// TIA Portal V18 export
TYPE "LGasp_typeBufferQuote"
// stored: IsFailsafeCompliant false
   STRUCT
      ID : DInt;
      n_piece : DInt;   // numero del pezzo a cui fa riferimento la quota
      general : "LGasp_typeArticoloGenerale";
      quota : "LGasp_typeQuota";
      quotaordinata : Bool;   // Quota ordinata da algoritmo riordino
   END_STRUCT;
END_TYPE
